// TwinCAT 3 PLC project PLCSim
// ProgramVersion: 3.1.4022.4
// libraries:
//   Tc2_Standard, * (Beckhoff Automation GmbH)
//   Tc2_System, * (Beckhoff Automation GmbH)
//   Tc3_Module, * (Beckhoff Automation GmbH)
//   VisuSymbols,3.5.10.0,System
// project tree:
//   / GlobalTextList.TcGTLO, PlcTask.TcTTO, Visualization Manager.TcVMO (not stored)
//   GVLs/ GVL.TcGVL
//   POUs/ AGV.TcPOU, MAIN.TcPOU, Process.TcPOU
//   POUs/Operation/ OperationPRG.TcPOU
//   VISUs/ AGVSimulator.TcVIS

CONFIGURATION PLCSim
    RESOURCE PLC ON TwinCAT3
        TASK PlcTask(INTERVAL := T#20ms, PRIORITY := 20);
        PROGRAM MAIN WITH PlcTask : MAIN;
    END_RESOURCE
END_CONFIGURATION

// ---- GVLs/GVL.TcGVL
{attribute 'qualified_only'}
VAR_GLOBAL
//Output from process to PLC
	qxAGVStrobe		AT %Q*:	BOOL;	(* AGV strobe signal *)
	qiAtPos			AT %Q*:	INT;	(* Actual position of AGV *)
	
//Input to process from PLC
	ixPLCStrobe		AT %I*:	BOOL;	(* PLC strobe signal *)
	iiGotoPos		AT %I*:	INT;	(* Target position for AGV *)
	ixStartButton   AT %I*: BOOL;   (* Start Button*)
	ixStopButton   	AT %I*: BOOL;   (* Stop Button*)
	ixResetButton   AT %I*: BOOL;   (* Reset Button*)
	
// Additional global variables 
	qxAGVMoving     AT %Q*: BOOL;   (* AGV Moving*)
	qxAGVLoc        AT %Q*: STRING; (* AGV Location*)
END_VAR

// ---- POUs/MAIN.TcPOU
PROGRAM MAIN
VAR
END_VAR

Process();
OperationPRG();

END_PROGRAM

// ---- POUs/Process.TcPOU
PROGRAM Process
VAR
	fbAGV: AGV;
END_VAR

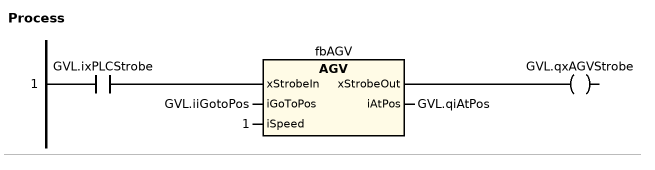
// NETWORK 1
fbAGV(xStrobeIn := GVL.ixPLCStrobe, iGoToPos := GVL.iiGotoPos, iSpeed := 1, iAtPos => GVL.qiAtPos); // AGV
GVL.qxAGVStrobe := fbAGV.xStrobeOut;

END_PROGRAM

// ---- POUs/AGV.TcPOU
FUNCTION_BLOCK AGV

VAR_INPUT
	xStrobeIn:		BOOL;	(* strobe in *)
	iGoToPos:		INT;	(* input go to position *)
	iSpeed:			INT;	(* AGV speed *)
END_VAR

VAR_OUTPUT
	xStrobeOut:		BOOL;	(* strobe out *)
	iAtPos:			INT;	(* output at pos *)
END_VAR

VAR
	iPhase:		 	INT;	(* phase in AGV handshake *)

	iGoToPosOld: 	INT;	(* previous cycle value *)
	iGoToReceived: 	INT;	(* saved value at rising edge of strobe in *)
	iGoTo:			INT;	(* set target value and start move *)
	iGoToPos_X: 	INT;	(* target X value *)
	iGoToPos_Y: 	INT;	(* target Y value *)
	iAtPos_X: 		INT;	(* actual X value *)
	iAtPos_Y: 		INT;	(* actual Y value *)
	iPos: 			INT;	(* actual pos, if any *)

	xError: 		BOOL;	(* AGV in error state *)

	fbStrobeOutR1: 	TON;	(* rising edge of strobe out when received message *)
	fbStrobeOutF1: 	TON;	(* falling edge of strobe out when received message *)
	fbStrobeOutR2: 	TON;	(* rising edge of strobe out when send message is set *)
	fbStrobeOutF2: 	TON;	(* falling edge of strobe out when send message is set *)

(* Define all Pos in X and Y *)
	iAGVPosHome_X: 	INT := 500;
	iAGVPosHome_Y: 	INT := 300;
	iAGVPosA_X: 	INT := 800;
	iAGVPosA_Y: 	INT := 0;
	iAGVPosB_X: 	INT := 800;
	iAGVPosB_Y: 	INT := 600;
	iAGVPosC_X: 	INT := 200;
	iAGVPosC_Y: 	INT := 600;
	iAGVPosD_X: 	INT := 200;
	iAGVPosD_Y: 	INT := 0;
	iAGVPosError_X: INT := 0;
	iAGVPosError_Y: INT := 300;
END_VAR

// Function Block AGV
// 20190118 v2_0 Bo Svensson University West

CASE iPhase OF
	(* ---- Handshake at receiving order ---- *)
0:		(* read old value of goto pos at rising edge of PLC strobe *)
	IF xStrobeIn AND (iGoToPosOld <> 0) AND ( iGoToPosOld <> iPos) THEN
		iGoToReceived := iGoToPosOld;
		iPhase := 10;
	END_IF

10:		(* send AGV strobe after read delay, indicate order received *)
	IF fbStrobeOutR1.Q THEN
		xStrobeOut := TRUE;
		iPhase :=20;
	ELSIF NOT xStrobeIn THEN
		xError := TRUE;
		iPhase := 500;
	END_IF

20:		(* wait for end of PLC strobe*)
	IF NOT xStrobeIn THEN
		iPhase := 30;
	END_IF

30:		(* send AGV ack after delay, indicate read order ended and activate AGV motion*)
	IF fbStrobeOutF1.Q THEN
		xStrobeOut := FALSE;
		iGoTo := iGoToReceived;
		iPhase := 40;
	ELSIF  xStrobeIn THEN
		xError := TRUE;
		iPhase := 500;
	END_IF

	(* --- AGV moves and finally reach target ---- *)
40:		(* set iAtPos when AGV stop moving *)
	IF ((iPos = iGoTo) AND (iGoTo <> 0)) OR (iGoTo = 6) THEN
		iAtPos := iPos;
		iPhase := 50;
	ELSIF (xStrobeIn AND (iGoToPosOld = 6))  THEN	(* instantly stop *)
		iGoToReceived := 6;
		iPhase := 10;
	ELSIF (xStrobeIn AND NOT (iGoToPosOld = 6))  THEN
		xError := TRUE;
		iPhase := 500;
	END_IF

	(* --- Handshake at answer --- *)
50:		(* send AGV strobe after delay, indicate target reached *)
	IF fbStrobeOutR2.Q THEN
		xStrobeOut := TRUE;
		iPhase := 60;
	ELSIF xStrobeIn THEN
		xError := TRUE;
		iPhase := 500;
	END_IF

60:		(* wait for PLC strobe *)
	IF  xStrobeIn AND (iGoToPosOld = 0) THEN
		iPhase := 70;
	END_IF

70:		(* remove AGV strobe and at pos after delay, indicating answer ready *)
	IF fbStrobeOutF2.Q THEN
		xStrobeOut := FALSE;
		iAtPos := 0;
		iPhase := 80;
	ELSIF NOT xStrobeIn THEN
		xError := TRUE;
		iPhase := 500;
	END_IF

80:		(* wait for end of PLC strobe *)
	IF  NOT xStrobeIn THEN
		iPhase := 0;
	END_IF

	(* --- Error state --- *)
500: 	(* goto error and do nothing more *)
	iGoTo := 100;
END_CASE

(* all timer block for iPhase states *)
fbStrobeOutR1(IN := xStrobeIn AND (iPhase = 10), PT := T#1S);
fbStrobeOutF1(IN := NOT xStrobeIn AND (iPhase = 30), PT := T#1S);
fbStrobeOutR2(IN := NOT xStrobeIn AND (iPhase = 50), PT := T#1S);
fbStrobeOutF2(IN := xStrobeIn AND (iPhase = 70), PT := T#1S);


(* ---- Set goto X and Y pos and move AGV ---- *)
CASE iGoTo OF
0:	(* Do nothing *)
	iGoToPos_X := iGoToPos_X;
	iGoToPos_Y := iGoToPos_Y;

1:	(* GoToHome *)
	iGoToPos_X := iAGVPosHome_X;
	iGoToPos_Y := iAGVPosHome_Y;

2:	(* GoToA *)
	iGoToPos_X := iAGVPosA_X;
	iGoToPos_Y := iAGVPosA_Y;

3:	(* GoToB *)
	iGoToPos_X := iAGVPosB_X;
	iGoToPos_Y := iAGVPosB_Y;

4:	(* GoToC *)
	iGoToPos_X := iAGVPosC_X;
	iGoToPos_Y := iAGVPosC_Y;

5:	(* GoToD *)
	iGoToPos_X := iAGVPosD_X;
	iGoToPos_Y := iAGVPosD_Y;

6:	(* Stop instantly *)
	iGoToPos_X := iAtPos_X;
	iGoToPos_Y := iAtPos_Y;

ELSE	(* GoToError *)
	iAtPos_X := iAGVPosError_X;
	iAtPos_Y := iAGVPosError_Y;
	xError := TRUE;
END_CASE


(* ---- AGV motion ---- *)
IF iAtPos_X < iGoToPos_X THEN
	iAtPos_X := iAtPos_X + iSpeed;
ELSIF iAtPos_X > iGoToPos_X THEN
	iAtPos_X := iAtPos_X - iSpeed;
END_IF

IF iAtPos_Y < iGoToPos_Y THEN
	iAtPos_Y := iAtPos_Y + iSpeed;
ELSIF iAtPos_Y > iGoToPos_Y THEN
	iAtPos_Y := iAtPos_Y - iSpeed;
END_IF


(* ---  AGV actual position --- *)
IF iAtPos_X = iAGVPosHome_X AND iAtPos_Y = iAGVPosHome_Y THEN
	iPos := 1;		(* Pos Home *)
ELSIF iAtPos_X = iAGVPosA_X AND iAtPos_Y = iAGVPosA_Y THEN
	iPos := 2;		(* Pos A *)
ELSIF iAtPos_X = iAGVPosB_X AND iAtPos_Y = iAGVPosB_Y THEN
	iPos := 3;		(* Pos B *)
ELSIF iAtPos_X = iAGVPosC_X AND iAtPos_Y = iAGVPosC_Y THEN
	iPos := 4;		(* Pos C *)
ELSIF iAtPos_X = iAGVPosD_X AND iAtPos_Y = iAGVPosD_Y THEN
	iPos := 5;		(* Pos D *)
ELSIF iGoTo = 6 THEN
	iPos := 6;		(* Instant stop not at any pos *)
ELSE
	iPos := 0;		(* Not at any Pos *)
END_IF


(* save goto pos input value to next turn *)
iGoToPosOld := iGoToPos;

END_FUNCTION_BLOCK

// ---- POUs/Operation/OperationPRG.TcPOU
PROGRAM OperationPRG
VAR
	mxPosA 		  : BOOL;
	mxPosB 		  : BOOL;
	mxPosC 		  : BOOL;
	mxPosD 		  : BOOL;
	mxPosHome 	  : BOOL;
	mxPosInit 	  : BOOL;

END_VAR

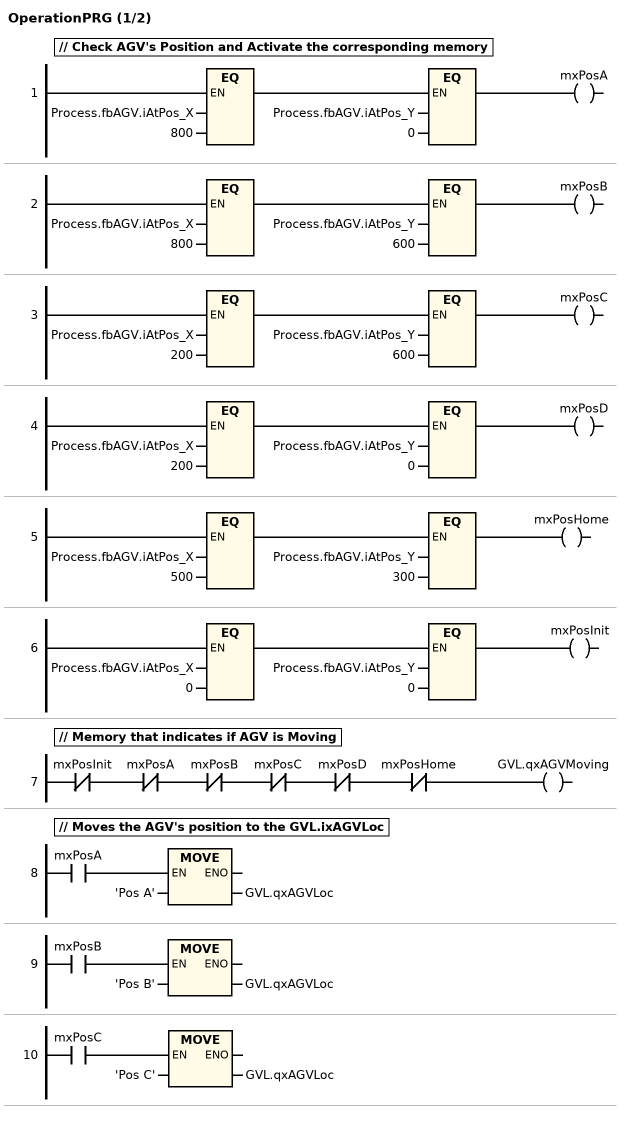
// NETWORK 1
// label: // Check AGV's Position and Activate the corresponding memory
mxPosA := Process.fbAGV.iAtPos_X = 800 AND Process.fbAGV.iAtPos_Y = 0;

// NETWORK 2
mxPosB := Process.fbAGV.iAtPos_X = 800 AND Process.fbAGV.iAtPos_Y = 600;

// NETWORK 3
mxPosC := Process.fbAGV.iAtPos_X = 200 AND Process.fbAGV.iAtPos_Y = 600;

// NETWORK 4
mxPosD := Process.fbAGV.iAtPos_X = 200 AND Process.fbAGV.iAtPos_Y = 0;

// NETWORK 5
mxPosHome := Process.fbAGV.iAtPos_X = 500 AND Process.fbAGV.iAtPos_Y = 300;

// NETWORK 6
mxPosInit := Process.fbAGV.iAtPos_X = 0 AND Process.fbAGV.iAtPos_Y = 0;

// NETWORK 7
// label: // Memory that indicates if AGV is Moving
GVL.qxAGVMoving := NOT mxPosInit AND NOT mxPosA AND NOT mxPosB AND NOT mxPosC AND NOT mxPosD AND NOT mxPosHome;

// NETWORK 8
// label: // Moves the AGV's position to the GVL.ixAGVLoc
IF mxPosA THEN GVL.qxAGVLoc := 'Pos A'; END_IF

// NETWORK 9
IF mxPosB THEN GVL.qxAGVLoc := 'Pos B'; END_IF

// NETWORK 10
IF mxPosC THEN GVL.qxAGVLoc := 'Pos C'; END_IF

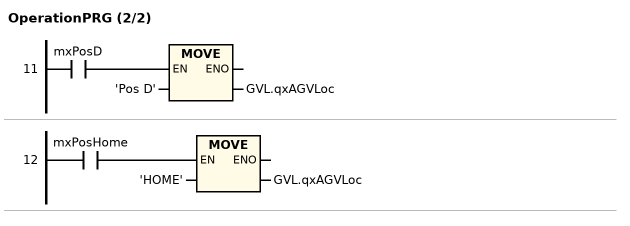
// NETWORK 11
IF mxPosD THEN GVL.qxAGVLoc := 'Pos D'; END_IF

// NETWORK 12
IF mxPosHome THEN GVL.qxAGVLoc := 'HOME'; END_IF

END_PROGRAM

// ---- GlobalTextList.TcGTLO
TEXTLIST GlobalTextList
  546 = 'AGV'
  738 = 'ERROR'
  838 = 'HOME'
  505 = 'Pos A'
  284 = 'Pos AD'
  908 = 'Pos B'
  412 = 'Pos C'
  547 = 'Pos D'
  315 = 'University West'
  428 = 'Ver 2.0'
END_TEXTLIST

// ---- VISUs/AGVSimulator.TcVIS
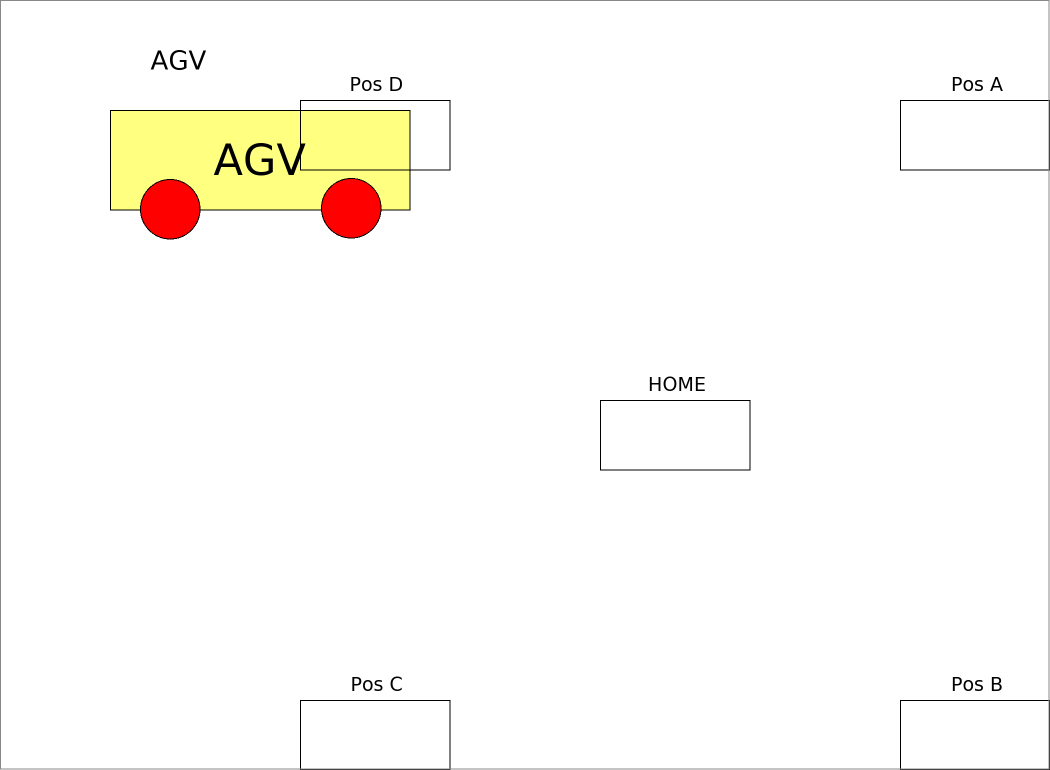
VISUALIZATION AGVSimulator  // 1050x770
    Group (110,110 130x50)
        p3560616238: Process.fbAGV.iAtPos_X
        p2738717112: Process.fbAGV.iAtPos_Y
        RoundedRectangle (0,0 300x100), "AGV"
        Ellipse (30,69 60x60)
        Ellipse (211,68 60x60)
    RoundedRectangle (300,100 150x70)
    RoundedRectangle (900,100 150x70)
    RoundedRectangle (600,400 150x70)
    RoundedRectangle (900,700 150x70)
    RoundedRectangle (300,700 150x70)
    Rectangle (330,670 94x29), "Pos C"
    Rectangle (930,670 94x29), "Pos B"
    Rectangle (930,70 94x29), "Pos A"
    Rectangle (330,70 93x29), "Pos D"
    Rectangle (630,370 94x29), "HOME"
    Rectangle (130,370 94x29), "ERROR", invisible if: NOT Process.fbAGV.xError
    Rectangle (91,46 175x29), "AGV"
    RoundedRectangle (107,356 144x54), invisible if: Process.fbAGV.xError
END_VISUALIZATION
